FUNCTION_BLOCK ColorDetect (* Composite Function Block Type *)
  (* Standard: 61499-2 *)
  (* Version 0.0, 9/28/2018, dmidro, nxtControl GmbH, template *)
  PACKAGE Main;
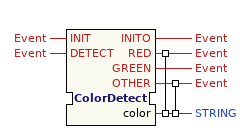
  EVENT_INPUT
    INIT; (* Initialization Request *)
    DETECT; (* Write data request event *)
  END_EVENT
  EVENT_OUTPUT
    INITO; (* Initialization Confirm *)
    RED WITH color; (* Event Output *)
    GREEN; (* Event Output *)
    OTHER WITH color; (* Event output *)
  END_EVENT
  VAR_OUTPUT
    color : STRING; (* Data read with every IND event *)
  END_VAR
  FBS
    FB1 : TCPIO(QI := TRUE, PORT := UDP:10011;192.168.0.77:9013, DATAOUT := CHECK);
    FB2 : COMPARE_10593E80BE744DDAF(IN1 := 'RED'); {SET_ATTRIBUTE(Configuration.GenericFBType.InterfaceParams, Runtime.Standard#CNT:=2;IN${CNT$}:STRING)}
    FB4 : COMPARE_10593E80BE744DDAF(IN1 := 'GREEN'); {SET_ATTRIBUTE(Configuration.GenericFBType.InterfaceParams, Runtime.Standard#CNT:=2;IN${CNT$}:STRING)}
    FB6 : AND_88A3DD8EC65DD11C; {SET_ATTRIBUTE(Configuration.GenericFBType.InterfaceParams, Runtime.Standard#CNT:=2;OUT:BOOL)}
    FB7 : E_REND;
    FB3 : E_PERMIT;
    FB5 : E_PERMIT;
    FB8 : E_PERMIT;
    FB10 : E_CTU(PV := 2);
    FB9 : E_PERMIT;
    FB11 : E_DELAY(DT := T#3s);
  END_FBS
  EVENT_CONNECTIONS
    FB1.INITO TO INITO;
    INIT TO FB1.INIT;
    DETECT TO FB11.START;
    FB9.EO TO FB2.REQ;
    FB9.EO TO FB4.REQ;
    FB2.CNF TO FB7.EI1;
    FB4.CNF TO FB7.EI2;
    FB7.EO TO FB6.REQ;
    FB2.CNF TO FB3.EI;
    FB3.EO TO RED;
    FB4.CNF TO FB5.EI;
    FB5.EO TO GREEN;
    FB6.CNF TO FB8.EI;
    FB8.EO TO OTHER;
    FB10.CUO TO FB9.EI;
    FB1.IND TO FB10.CU;
    DETECT TO FB1.REQ;
    DETECT TO FB10.R;
    FB11.EO TO FB1.REQ;
    FB1.CNF TO FB1.ACK;
  END_CONNECTIONS
  DATA_CONNECTIONS
    FB1.DATAIN TO color;
    FB1.DATAIN TO FB2.IN2;
    FB1.DATAIN TO FB4.IN2;
    FB2.NE TO FB6.IN1;
    FB4.NE TO FB6.IN2;
    FB2.EQ TO FB3.PERMIT;
    FB4.EQ TO FB5.PERMIT;
    FB6.OUT TO FB8.PERMIT;
    FB10.Q TO FB9.PERMIT;
  END_CONNECTIONS
END_FUNCTION_BLOCK
